(* CoDeSys 2.3.9.35 project: EX02.pro *)
(* Author: Altus *)
(* Libraries: DU35x.lib 7.7.11 15:59:13, Navigation.lib 15.7.11 10:06:00, SysLibTargetVisu.lib 26.11.08 09:53:28, Standard.lib 26.11.08 09:46:20, Iecsfc.lib 26.11.08 09:46:14, SYSLIBCALLBACK.LIB 26.11.08 09:53:30 *)

(* PLC configuration (modules and I/O channels)
COM1 [COM1] node 0, in %IB0 out %QB0 {BaudRate = 115200; Paridade = Sem Paridade; StopBits = 1 Stop Bit; Modem = Sem RTS/CTS; Delay = 5}
  MToolIEC [Codesys] node 0, in %IB0 out %QB0
Relação MODBUS [Relacao] node 0, in %IB0 out %QB0 {EnderecoModbus = 69; HoldRegisters = 3; OperandoModbus = 8; FuncaoModbus = Read Holding Registers; Polling = 1000; OperandoCodesys = %MW0; TipoCodesys = %MX}
Relação MODBUS [Relacao] node 1, in %IB0 out %QB0 {EnderecoModbus = 69; HoldRegisters = 1; OperandoModbus = 11; FuncaoModbus = Write Single Register; Polling = 100; OperandoCodesys = %MW3; TipoCodesys = %MX}
Barramento [Barramento] node 1, in %IB0 out %QB0
  Entradas [Entradas] node 0, in %IB0 out %QB0
    Entradas Digitais 0 [Entradas0] node 0, in %IW0 out %QB0
      I00 AT %IX0.0 [BitInput] I0.0
      I01 AT %IX0.1 [BitInput] I0.1
      I02 AT %IX0.2 [BitInput] I0.2
      I03 AT %IX0.3 [BitInput] I0.3
      I04 AT %IX0.4 [BitInput] I0.4
      I05 AT %IX0.5 [BitInput] I0.5
      I06 AT %IX0.6 [BitInput] I0.6
      I07 AT %IX0.7 [BitInput] I0.7
      I08 AT %IX0.8 [BitInput] I0.8
    Entradas Digitais 1 [Entradas1] node 0, in %IW1 out %QB0
      I10 AT %IX1.0 [BitInput] I1.0
      I11 AT %IX1.1 [BitInput] I1.1
      I12 AT %IX1.2 [BitInput] I1.2
      I13 AT %IX1.3 [BitInput] I1.3
      I14 AT %IX1.4 [BitInput] I1.4
      I15 AT %IX1.5 [BitInput] I1.5
      I16 AT %IX1.6 [BitInput] I1.6
      I17 AT %IX1.7 [BitInput] I1.7
      I18 AT %IX1.8 [BitInput] I1.8
    Entradas Digitais 2 [Entradas2] node 0, in %IW2 out %QB0
      I20 AT %IX2.0 [BitInput] I2.0
      I21 AT %IX2.1 [BitInput] I2.1
    Entradas Analógicas [EntradaAnalogica] node 0, in %IW4 out %QB0
      AI0 AT %IW4 [WordInput] AI0 {TipoAnalogica = Channel Disable; FiltroAnalogica = Filter 0 - AI=2ms  / AV=90ms; FundoEscala = 0}
      AI1 AT %IW5 [WordInput] AI1 {TipoAnalogica = Channel Disable; FiltroAnalogica = Filter 0 - AI=2ms  / AV=90ms; FundoEscala = 0}
      AI2 AT %IW6 [WordInput] AI2 {TipoAnalogica = Channel Disable; FiltroAnalogica = Filter 0 - AI=2ms  / AV=90ms; FundoEscala = 0}
      AI3 AT %IW7 [WordInput] AI3 {TipoAnalogica = Channel Disable; FiltroAnalogica = Filter 0 - AI=2ms  / AV=90ms; FundoEscala = 0}
    Entradas Rápidas [EntradasRapidas] node 1, in %IB16 out %QB0
      Bloco 0 [Bloco0] node 0, in %IB16 out %QB0
        Desabilitado [DesabilitadoBloco0] node 0, in %IB16 out %QB0
      Bloco 1 [Bloco1] node 1, in %IB16 out %QB0
        Desabilitado [DesabilitadoBloco1] node 0, in %IB16 out %QB0
      Entrada Configuravél Bloco 0 [EntradaConfiBloco0] node 2, in %IB16 out %QB0
        Contador 0 [EntradaConfContador0] node 0, in %IB16 out %QB0 {EntradaConfiguravelContador = Disable}
      Entrada Configuravél Bloco 1 [EntradaConfiBloco1] node 3, in %IB16 out %QB0
        Contador 2 [EntradaConfContador2] node 0, in %IB16 out %QB0 {EntradaConfiguravelContador = Disable}
  Saídas [Saidas] node 1, in %IB13 out %QB0
    Saídas Digitais 0 [Saidas0] node 0, in %IW0 out %QW0
      Q00 AT %QX0.0 [BitOutput] Q0.0
      Q01 AT %QX0.1 [BitOutput] Q0.1
      Q02 AT %QX0.2 [BitOutput] Q0.2
      Q03 AT %QX0.3 [BitOutput] Q0.3
      Q04 AT %QX0.4 [BitOutput] Q0.4
      Q05 AT %QX0.5 [BitOutput] Q0.5
      Q06 AT %QX0.6 [BitOutput] Q0.6
      Q07 AT %QX0.7 [BitOutput] Q0.7
    Saídas Digitais 1 [Saidas1] node 0, in %IW0 out %QW1
      Q10 AT %QX1.0 [BitOutput] Q1.0
      Q11 AT %QX1.1 [BitOutput] Q1.1
      Q12 AT %QX1.2 [BitOutput] Q1.2
      Q13 AT %QX1.3 [BitOutput] Q1.3
      Q14 AT %QX1.4 [BitOutput] Q1.4
      Q15 AT %QX1.5 [BitOutput] Q1.5
      Q16 AT %QX1.6 [BitOutput] Q1.6
      Q17 AT %QX1.7 [BitOutput] Q1.7
    Saídas Analógicas [SaidaAnalogica] node 0, in %IW0 out %QW3
      AO0 AT %QW3 [WordOutput] AO0 {TipoAnalogica = Channel Disable; FundoEscala = 0}
      AO1 AT %QW4 [WordOutput] AO1 {TipoAnalogica = Channel Disable; FundoEscala = 0}
    Saídas Rápidas [SaidasRapidas] node 1, in %IB0 out %QB10
      Saída Rápida 0 Desabilitada [DesabilitadoF0] node 0, in %IB0 out %QB10
      Saída Rápida 1 Desabilitada [DesabilitadoF1] node 1, in %IB0 out %QB10
    Saídas Comum de Contador [SaidasContador] node 2, in %IB0 out %QB10
      Saída do Bloco 0 Desabilitada [DesabilitadoSaidaBloco0] node 0, in %IB0 out %QB10
      Saída do Bloco 1 Desabilitada [DesabilitadoSaidaBloco1] node 1, in %IB0 out %QB10
Eventos Externos [Eventos] node 2, in %IB13 out %QB6
  Evento Temporizado [TimerEvent] node 0, in %IB13 out %QB6 {Intervalo = 10}
*)

(* Task configuration *)
TASK PRINCIPAL (PRIORITY := 1, INTERVAL := T#1ms);
	PLC_PRG();
END_TASK
TASK NAVIGATION (PRIORITY := 1, INTERVAL := T#20ms);
	NAVEGA();
END_TASK
TASK VISUALIZATION (PRIORITY := 1, INTERVAL := T#500ms);
	MAINTARGETVISU_PAINT_CODE
END_TASK
TASK KEYBOARD_USAGE (PRIORITY := 1, INTERVAL := T#20ms);
	MAINTARGETVISU_INPUT_CODE
END_TASK

(* POU PLC_PRG, ST *)
PROGRAM PLC_PRG
VAR
	TEMP AT %MW0 : WORD;
	UMID AT %MW1 : WORD;
	PO AT %MW2 : WORD;
	TEMP_REAL : REAL;
	UMID_REAL: REAL;
	PO_REAL : REAL;
	UN AT %MW3 : WORD;
	F4 : BOOL;
END_VAR
TEMP_REAL := WORD_TO_REAL(TEMP) / 10;
UMID_REAL := WORD_TO_REAL(UMID) / 10;
PO_REAL := WORD_TO_REAL(PO) / 10;

IF F4 = TRUE THEN
	UN := 1;
ELSE
	UN := 0;
END_IF
END_PROGRAM

(* POU NAVEGA, ST *)
PROGRAM NAVEGA
VAR
	ControleTelas : NAVIGATION;
	ListaTelas 	: ARRAY [0..30] OF STRING(10);
END_VAR
(* Adiciona a tela MAIN como tela principal *)
ListaTelas[0] := 'MAIN';

(* Ativa o controle automático de navegação somente pelo teclado *)
ControleTelas(ENABLE_UPDW := FALSE, VISU_LIST := ListaTelas, UP := FALSE , DOWN := FALSE);
END_PROGRAM

(* Visualisation MAIN
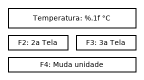
rectangle at (0,0)-(128,20): text "Temperatura: %.1f °F"; shows PLC_PRG.TEMP_REAL
rectangle at (0,27)-(60,42): text "F2: 2a Tela"
rectangle at (68,27)-(128,42): text "F3: 3a Tela"
rectangle at (0,49)-(128,64): text "F4: Muda unidade"
rectangle at (0,0)-(128,20): text "Temperatura: %.1f °C"; shows PLC_PRG.TEMP_REAL; invisible if PLC_PRG.F4
*)

(* Visualisation SEG
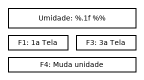
rectangle at (0,0)-(128,20): text "Umidade: %.1f %%"; shows PLC_PRG.UMID_REAL
rectangle at (0,27)-(60,42): text "F1: 1a Tela"
rectangle at (68,27)-(128,42): text "F3: 3a Tela"
rectangle at (0,49)-(128,64): text "F4: Muda unidade"
*)

(* Visualisation TERC
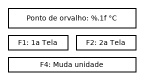
rectangle at (0,0)-(128,20): text "Ponto de orvalho: %.1f °F"; shows PLC_PRG.PO_REAL
rectangle at (0,27)-(60,42): text "F1: 1a Tela"
rectangle at (68,27)-(128,42): text "F2: 2a Tela"
rectangle at (0,49)-(128,64): text "F4: Muda unidade"
rectangle at (0,0)-(128,20): text "Ponto de orvalho: %.1f °C"; shows PLC_PRG.PO_REAL; invisible if PLC_PRG.F4
*)
